// TIA Portal V20 export
DATA_BLOCK "ET500SP_509"   // DB233
// stored: MemoryReserve 100
   VAR
      "SP509.00 UNWINDER EPCC01 INTERKOCK" : Bool;
      "SP509.01 UNWINDER EPCC02 INTERLOCK" : Bool;
      "SP509.02 UNWINDER EPCC03 INTERLOCK" : Bool;
      SPARE1 : Bool;
      SPARE2 : Bool;
      SPARE3 : Bool;
      SPARE4 : Bool;
      SPARE5 : Bool;
   END_VAR
BEGIN
END_DATA_BLOCK
